// This function has been automatically generated from the project information.
{attribute 'signature_flag' := '1073741824'}
{attribute 'TcGenerated'}
{attribute 'no-analysis'}
FUNCTION F_GetCompany : WSTRING
VAR_INPUT
	
END_VAR

F_GetCompany := "ekvip automation GmbH";

END_FUNCTION

(* stored: Version 1.1.0.1
   POU F_GetCompany: Id {d4859e3c-c274-4db2-a2ad-bd1020f7984e}, SpecialFunc None *)
